{attribute 'GeneratedUsingTerminal: EKM1101-0000-0016'}
{attribute addProperty BoxType "EKM1101-0000-0016"}
{attribute addProperty Id "ValueAT %I*INT2"}
{attribute addProperty CRC "2162654570"}
{attribute addProperty Size "2"}
TYPE MMS_Acceleration_Z_Axis_80E77D6A :
STRUCT
	{attribute addProperty Name "Value"}
	Value AT %I* : INT;
END_STRUCT
END_TYPE

(* stored: Version 1.2.0.0, ProductVersion 3.1.4024.9
   DUT MMS_Acceleration_Z_Axis_80E77D6A: Id {2fb3a0d6-b96e-4329-b20d-d45cb9b1c0e9} *)
